FUNCTION_BLOCK Skill_Position_anfahren_erweitert EXTENDS GrundstrukturSkill
VAR_INPUT 
	sProzessvariablen			:sRoboterProzessVariablen;
	bLimitTrig					:BOOL;
	bErreichtTrig				:BOOL;
END_VAR
VAR_OUTPUT
	sObjektvariablen			:sRoboterProzessVariablen;
END_VAR
VAR
	
END_VAR

// Fehlerüberwachung
IF bFehler THEN
	iState := 3;
END_IF

//_______________________________________________________________
// Reaktion auf Input-Variablen:
	// Starten
	fTrigger(CLK := bExecute);
	fSwitch(Set1 := fTrigger.Q);
	
	IF fSwitch.Q1 AND iSysState = 1 THEN
		bStarten := TRUE;
		fSwitch.RESET := TRUE;
	ELSE
		bStarten := FALSE;
		fSwitch.RESET := FALSE;
	END_IF

	// Stoppen
	IF iSysCommand = 3 THEN
		bStoppen := TRUE;
	ELSE 
		bStoppen := FALSE;
	END_IF

	// Resetten 
	IF iSysCommand = 4 THEN
		bResetten := TRUE;
	ELSE
		bResetten := FALSE;
	END_IF
	
	// Limit 
	IF bLimitTrig THEN
		bLimitReached := TRUE;
	ELSE
		bLimitReached := FALSE;
	END_IF
	// Erreicht
	IF bErreichtTrig THEN
		bTargetReached := TRUE;
	ELSE 
		bTargetReached := FALSE;
	END_IF
	

//_______________________________________________________________
// Zustandsmanagement
CASE iState OF 
0: 	// BEREIT
		// DO
		bDone := FALSE;	
	
		IF bStarten THEN
			IF ParameterError OR PositionError THEN
				bError := TRUE;
			ELSE	
				sObjektvariablen := sProzessvariablen;
				iSkillCommand := 1;																						// Starten des Objektes 
			END_IF		
		END_IF	
		
		IF iObjState = 3 THEN																					// Resetten von Startsignal
			bGestartet := TRUE;
		END_IF
			
		// TRANSITION	
		IF bGestartet THEN
			bGestartet := FALSE;
			iState := 1;																								// Objekt wurde gestartet
		END_IF
// _________________________________________________________________________________________________________________________
1: 	// LAUFEND
		// DO
		iSkillCommand := 0;
		bBusy := TRUE;																									// Skill wird ausgeführt
		
		
		IF bTargetReached OR bLimitReached THEN																			// Prüfen ob Prozessziel erreicht wurde
			iSkillCommand := 2;
		END_IF
		
		IF iObjState = 4 THEN																							// Objekt hat Prozess abgeschlossen
			bBusy := FALSE;																									// Skill wird nicht mehr ausgeführt			
			bObjektFertig := TRUE;																							// Objekt ist fertig und wieder bereit
		END_IF
		
		IF bStoppen THEN																							// Transition wenn System das Orbjekt stoppt
			bBusy := FALSE;																									// Skill wird nicht mehr ausgeführt
		END_IF
		
		IF bLimitReached AND iObjState = 5 THEN																			// Objekt wurde duch Skill gestoppt - LIMIT
			iSkillCommand := 0;																								// Zurücksetzen von Command																						// Zurücksetzen von Information	
			bBusy := FALSE;																									// Skill wird nicht mehr ausgeführt
			bLimitErreicht := TRUE;	
		END_IF
		
		IF bTargetReached AND iObjState = 5 THEN																			// Objekt wurde duch Skill gestoppt - LIMIT
			iSkillCommand := 0;																									// Zurücksetzen von Command
			bTargetReached := FALSE;																							// Zurücksetzen von Information	
			bBusy := FALSE;																										// Skill wird nicht mehr ausgeführt
			bWertErreicht := TRUE;	
		END_IF
			
		// TRANSITION 
		IF bObjektFertig THEN																							// Transition zu ABGESCHLOSSEN
			bObjektFertig := FALSE;																							// Skill wird nicht mehr ausgeführt
			iState := 2;																									// Objekt ist fertig und wieder bereit
		END_IF
		
		IF bGestoppt THEN																									// Transition zu BEREIT
			bGestoppt := FALSE;																							
			iState := 0;
		END_IF
		
		IF bLimitErreicht THEN																							// Transition zu LIMIT
			bLimitErreicht := FALSE;
			iState := 4;
		END_IF
		
		IF bWertErreicht THEN																							// Transition zu ERREICHT																						// Skill wird nicht mehr ausgeführt
			bWertErreicht := FALSE;
			iState := 5;
		END_IF
			
// _________________________________________________________________________________________________________________________			
2: 	// ABGESCHLOSSEN
		// DO																												// Skill wurde erfolgreich ausgeführt
		iSkillCommand := 3;
		bDone := TRUE;																										// Objekt resetten
		
		IF iObjState = 1 THEN
			iSkillCommand := 0;																								// Zurücksetzen von Command
			bSkillFertig := TRUE;											
		END_IF
			
		//  TRANSITION
		IF bSkillFertig THEN
			bSkillFertig := FALSE;																							// Zurücksetzen von Skill																																										// Resetten von Objekt
			iState := 0;
		END_IF
		
// _________________________________________________________________________________________________________________________
3: 	// FEHLER
		// DO 
		iSkillCommand := 0;	
		bDone := FALSE;
		bBusy := FALSE;
		
		IF ParameterError THEN
			// Setzen von ErrorID
		END_IF
		
		IF PositionError THEN
			// Setzen von ErrorID
		END_IF
		
		// TRANSITION
		IF bResetten THEN
			iState := 0;
		END_IF
		
// _________________________________________________________________________________________________________________________			
4: 	// LIMIT
		// DO 
		bLimit := TRUE;																									// Limit wurde erreicht
		iSkillCommand := 3;																								// Objekt resetten
		
		IF iObjState = 1 THEN																							// Objekt wurde geresettet
			iSkillCommand := 0;																								// Zurücksetzen von Command
			bDone := FALSE;																									// Zurücksetzen von Skill
			bResetten := TRUE;								
		END_IF
	
		// TRANSITION
		IF bResetten THEN
			bResetten := FALSE;
			bLimit := FALSE;																							// Zurücksetzen von Output-Variable
			iState := 0;
		END_IF
		
// _________________________________________________________________________________________________________________________
5: 	// ERREICHT		
		// DO 
		bDone := TRUE;																								// Skill wurde erfolgreich ausgeführt
		
		iSkillCommand := 3;																								// Objekt resetten
		
		IF iObjState = 1 THEN																							// Objekt wurde geresettet
			iSkillCommand := 0;																								// Zurücksetzen von Command
			bDone := FALSE;																									// Zurücksetzen von Skill
			bSkillFertig := TRUE;									
		END_IF
		
		// TRANSITION
		IF bSkillFertig THEN
			bSkillFertig := FALSE;
			iState := 0;
		END_IF

END_CASE

TRANSITION ParameterError:
IF sProzessvariablen.a = 0 OR sProzessvariablen.v = 0 THEN
	ParameterError := TRUE;
END_IF
END_TRANSITION

TRANSITION PositionError:
IF sProzessvariablen.q1 = 0 AND sProzessvariablen.q2 = 0 AND sProzessvariablen.q3 = 0 AND sProzessvariablen.q4 = 0 AND sProzessvariablen.q5 = 0 AND sProzessvariablen.q6 = 0 THEN
	PositionError := TRUE;
END_IF
END_TRANSITION

END_FUNCTION_BLOCK

(* stored: Version 1.1.0.1
   POU Skill_Position_anfahren_erweitert: Id {2c6ea44a-44bd-4f23-9af6-7ce31a275829}, SpecialFunc None
   Folder 01_Errors: Id {8ce5e8d8-c0c1-4f8d-a85b-0d4b99e34d4b}
   Transition ParameterError: Id {43f55938-bc4f-4bea-a68d-04049305a2eb}
   Transition PositionError: Id {58633fcd-fe1e-485e-8b85-3f801286f0bd} *)
